//==================================================================================================
//							Beckhoff Automation Poland
//									14.03.2023
//
// Code owner: TG
//
// Function block for processing digital inputs. 
// Includes filters, simulating and edges detection.
//
// Used libraries: 
//	Tc2_standard						|| 3.3.3.0
//
// Used FBs:
//
// Used DUTs:
//
//  v1.0	|| TC v 3.1.4024.40		|| First edition
//==================================================================================================
FUNCTION_BLOCK FB_DigitalInput_1

VAR_INPUT
	In 											: BOOL;
END_VAR

VAR
	
	bManual										: BOOL;	 // HMI
	bManualIn									: BOOL;	 // HMI
	{attribute 'hide'}
	_bCheckFS									: BOOL;
	{attribute 'hide'}
	_bIn	 									: BOOL;
	{attribute 'hide'}
	_bInRE										: BOOL;
	{attribute 'hide'}
	_bInFE										: BOOL;
	{attribute 'hide'}
	_tTimeOn									: TIME;
	{attribute 'hide'}
	_tTimeOff									: TIME;	
	{attribute 'hide'}
	_tTimeFS									: TIME;
	{attribute 'hide'}
	TimeFS										: TOF;	
	{attribute 'hide'}
	rtTrigger									: R_TRIG;
	{attribute 'hide'}
	ftTrigger									: F_TRIG;
END_VAR

{attribute 'monitoring' := 'variable'}
PROPERTY bCheckFS								: BOOL
GET
bCheckFS										:= _bCheckFS;
END_GET
SET
_bCheckFS										:= bCheckFS;
END_SET
END_PROPERTY

{attribute 'monitoring' := 'variable'}
PROPERTY bErrFS 								: BOOL							//Fail-safe error
GET
bErrFS											:= NOT TimeFS.Q AND bCheckFS;
END_GET
END_PROPERTY

{attribute 'monitoring' := 'variable'}
PROPERTY bIn 									: BOOL							//Processed input variable
GET
bIn												:= _bIn;
END_GET
SET
_bIn											:= bIn;
END_SET
END_PROPERTY

{attribute 'monitoring' := 'variable'}
PROPERTY bInFE 									: BOOL							//Falling edge detected
GET
bInFE											:= ftTrigger.Q;
END_GET
END_PROPERTY

{attribute 'monitoring' := 'variable'}
PROPERTY bInRE 									: BOOL							//Rising edge detected
GET
bInRE											:= rtTrigger.Q;
END_GET
END_PROPERTY

METHOD Filter 									: BOOL							//Activation and disable filter
VAR_INST
	{attribute 'hide'}
	TimeON										: TON;
	{attribute 'hide'}
	TimeOFF										: TOF;	
END_VAR
TimeON(IN := In, PT := tTimeON);
TimeOFF(IN := TimeON.Q, PT := tTimeOff);

bIn												:= TimeOFF.Q;
END_METHOD

METHOD FilterTrig 								: BOOL						//Activation and disable filter with edges detection
Filter();		
RTrig();
FTrig();
END_METHOD

METHOD FS 										: BOOL								// Fail-safe detection timer
VAR_INST
	{attribute 'hide'}
	bLastIn										: BOOL;	
END_VAR
TimeFS(IN := bLastIn <> In, PT := tTimeFS);	

bLastIn											:= In;
END_METHOD

METHOD PRIVATE FTrig 							: BOOL							// Falling edge detection
ftTrigger(CLK := bIn);
END_METHOD

METHOD Manual 									: BOOL							//Manually controlled input
IF bManual THEN
	ManualEx(bIn := bManualIn);
END_IF
END_METHOD

METHOD ManualEx 									: BOOL							//Manually controlled input
VAR_INPUT
	bIn												: BOOL;
END_VAR
bCheckFS										:= FALSE;
bIn												:= bIn;
END_METHOD

METHOD ManualExTrig 								: BOOL						//Manually controlled input with edges detection
VAR_INPUT
	bManual											: BOOL;
	bIn												: BOOL;
END_VAR
ManualEx(bIn := bManualIn);		
RTrig();
FTrig();
END_METHOD

METHOD ManualTrig 								: BOOL						//Manually controlled input with edges detection
Manual();		
RTrig();
FTrig();
END_METHOD

METHOD Raw 										: BOOL							// Raw value
bIn												:= In;
END_METHOD

METHOD PRIVATE RTrig 							: BOOL							//Rising edge detection
rtTrigger(CLK := bIn);
END_METHOD

{attribute 'monitoring' := 'variable'}
PROPERTY tTimeFS 								: TIME							//fail-safe control time [ms]
GET
tTimeFS											:= _tTimeFS;
END_GET
SET
_tTimeFS										:= tTimeFS;
END_SET
END_PROPERTY

{attribute 'monitoring' := 'variable'}
PROPERTY tTimeOff 								: TIME						//disabling filter time [ms]
GET
tTimeOff										:= _tTimeOff;
END_GET
SET
_tTimeOff										:= tTimeOff;
END_SET
END_PROPERTY

{attribute 'monitoring' := 'variable'}
PROPERTY tTimeOn 								: TIME							//activation delay time [ms]
GET
tTimeOn											:= _tTimeOn;
END_GET
SET
_tTimeOn									:= tTimeOn;
END_SET
END_PROPERTY

END_FUNCTION_BLOCK

(* stored: Version 1.2.0.0, ProductVersion 3.1.4026.13, FileIdentifier 7626e5107441b41d94db2a6193ae224fd8a48ef4, FileSignature 92d9ff8524188467986ec21e987c37701c4227f927e85dd97f08ae18791335f029163f058a98a79496dc4dc1783005971ef4ef0ce546ce0084fb30906b19d4991bb0e8e0043b5623478f5157cc54e5e7d4510b95d7022c77fbb33b6f5ac3f5afe578302b2e648302a6a166d035fe6533e3c63b35f816b61ed3bb00b4928c31c288fefa2caff7dedee6dd2ad99e384f07e24a98f1484adc3ba4aa1877c74a1f5503a2e11c83f9662112d3fa3f1727e32721e4cca6efe3b09376bbb6fffee0de49bfce0801b074345d0c3e8bc10cb14ee5f4d56c5dfbd05dfba465ae6f096b8bf06d9e5ba940fbfd8fc38744e3fe77962fe68aeddc1548f48c7c9ef741996a41b6
   POU FB_DigitalInput_1: Id {201a31fd-9202-4872-bce7-77aaa6c92b8a}, SpecialFunc None
   Folder Methods: Id {5327c176-4c7a-49c4-9946-8623f4a5cad3}
   Folder Properties: Id {88d8864f-1bee-4d2b-85c9-2c0ea005a8a6}
   Property bCheckFS: Id {9b29110d-cb15-4c45-ab0f-a7e80ec3af84}
   Get Get: Id {5823c3ff-990c-4953-afe9-cbb1b527fab3}
   Set Set: Id {df8c9745-8e93-4a9a-9307-78da2f32331f}
   Property bErrFS: Id {dc08ff1f-e997-43dd-bcf9-1eb2436def5a}
   Get Get: Id {e715f7d8-da55-4c12-b0ff-cc04fb0abe9c}
   Property bIn: Id {b36d442f-ae08-4db6-9b60-d9e5059bf25a}
   Get Get: Id {17f7c879-2fe3-491b-9699-9b2ef0b670cf}
   Set Set: Id {e5b5221f-f935-4231-bab9-87fed15485f0}
   Property bInFE: Id {e0ce7c23-2638-4b11-afa9-e83c15e7e3a3}
   Get Get: Id {bdca280e-40a1-48b3-ad33-58719eda63c2}
   Property bInRE: Id {fe54431a-1f1f-4a76-961e-e175cf9b45a5}
   Get Get: Id {bb771e0d-fe86-4aef-b3a3-faf8b0db9e91}
   Method Filter: Id {42a27112-e862-4857-bb64-871ffe6fa761}
   Method FilterTrig: Id {0ddf6db1-0696-4775-a3d7-f8f5a3eb0ea8}
   Method FS: Id {2cd94628-eca5-4c8c-91e6-37528bb35177}
   Method FTrig: Id {71963bea-9759-4e1c-8034-a278b57f7156}
   Method Manual: Id {4359c507-320c-48e1-9098-8e5c30699421}
   Method ManualEx: Id {a59de4d9-a93d-4360-a73f-526be35374a8}
   Method ManualExTrig: Id {cc421c79-0c4b-433b-83b1-517dd6cafca0}
   Method ManualTrig: Id {88c45762-ad82-40ca-a835-1fc0be34d7f7}
   Method Raw: Id {52115bd8-35ad-4a71-bf48-3fb2fda0de26}
   Method RTrig: Id {6cde64ff-87b4-4dd0-9354-5da03bb87e1a}
   Property tTimeFS: Id {3ceceddf-4c7f-4aa4-a00d-af7688e28701}
   Get Get: Id {30859558-8ad6-41c8-9f9b-8c3050259bb6}
   Set Set: Id {9b81f1d4-1190-4f1a-af2d-6ab7fa18f394}
   Property tTimeOff: Id {de9a41dc-d558-4c7d-b59a-a9452b9706e5}
   Get Get: Id {df0ccf55-dd99-4a6e-8d49-00e37546091d}
   Set Set: Id {55ed4bc9-77e1-4056-b502-b9dbeacf2f8a}
   Property tTimeOn: Id {fcae59d8-50fc-46fe-8d03-e4e6493004aa}
   Get Get: Id {bc4b331f-8c31-465c-bda1-0d5af7beb8ce}
   Set Set: Id {8be578ae-4654-4f96-8c1a-5dd96d36f8df} *)
